FUNCTION_BLOCK TEST_DWORD (* Test DWORD AND,OR,XOR *)
  (* Standard: 61131-3 *)
  (* Version 0.0, 2006-09-02, JHC, Holobloc Inc, Converted from TEST_BYTE. *)
  (* Compiler header: package fb.rt.test; *)
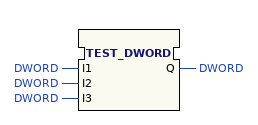
  VAR_INPUT
    I1 : DWORD;
    I2 : DWORD;
    I3 : DWORD;
  END_VAR
  VAR_OUTPUT
    Q : DWORD;
  END_VAR
  ALGORITHM REQ IN FBD:
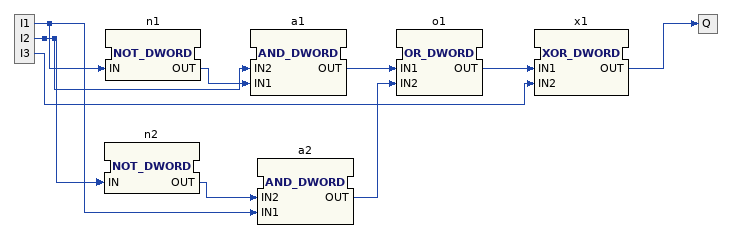
    FBS
      n1 : NOT_DWORD;
      n2 : NOT_DWORD;
      a1 : AND_DWORD;
      a2 : AND_DWORD;
      o1 : OR_DWORD;
      x1 : XOR_DWORD;
    END_FBS
    DATA_CONNECTIONS
      I1 TO n1.IN;
      I2 TO n2.IN;
      I2 TO a1.IN2;
      n2.OUT TO a2.IN2;
      n1.OUT TO a1.IN1;
      I1 TO a2.IN1;
      a1.OUT TO o1.IN1;
      a2.OUT TO o1.IN2;
      o1.OUT TO x1.IN1;
      I3 TO x1.IN2;
      x1.OUT TO Q;
    END_CONNECTIONS
  END_ALGORITHM
END_FUNCTION_BLOCK
